// TIA Portal V18 export
FUNCTION_BLOCK "Scen2_Diag"   // FB2, FBD
TITLE = demonstrates on one variable how to generate an Alarm for HMI
   VAR_INPUT
      ID : DInt;
      Port : Int;
      EV_ID : C_Alarm_s;
   END_VAR
   VAR_OUTPUT
      Error : Bool;
      Status : Word;
      DiagDeviceFB : "LIOLink_typeDiagnostics";
   END_VAR
   VAR
      Ret : Int;
      timestamp : Date_And_Time;
      data { S7_SetPoint := 'True'} : "LIOLink_3RB24_typeAll";
      IO_LINK_3RB24_300_400_Instance { S7_SetPoint := 'True'} : "LIOLink_3RB24";
      REQ : Bool;
      Done : Bool;
      busy : Bool;
      M3 : Bool;
      M2 : Bool;
      M1 : Bool;
      error_1 : Bool;
      IEC_Timer_0_Instance { S7_SetPoint := 'True'} : TP;
   END_VAR
   VAR_TEMP
      Error_temp_1 : Bool;
      Error_temp_2 : Bool;
      status_1 : DWord;
      status_2 : DWord;
   END_VAR
   VAR_TEMP   // added for the SCL form of the ladder/FBD networks
      _w1 : Bool;
   END_VAR
BEGIN

REGION Network 1
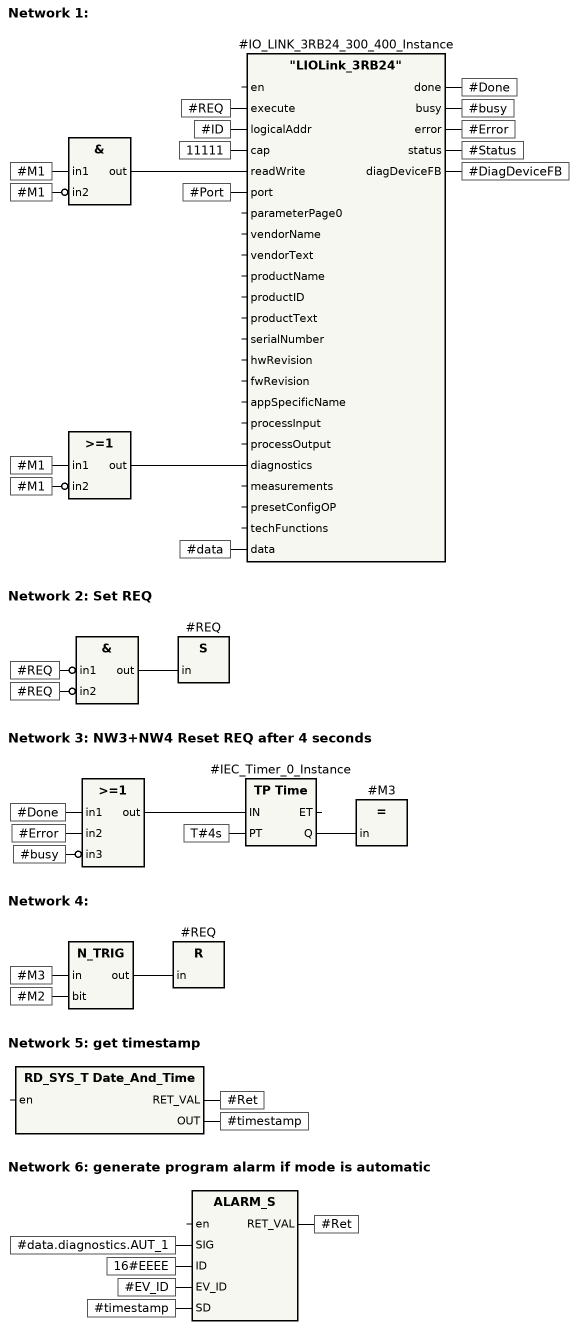
   #IO_LINK_3RB24_300_400_Instance(execute := #REQ,   // "LIOLink_3RB24"
                           logicalAddr := #ID,
                           cap := 11111,
                           readWrite := #M1 AND NOT #M1,
                           port := #Port,
                           diagnostics := #M1 OR NOT #M1,
                           data := #data,
                           done => #Done,
                           busy => #busy,
                           error => #Error,
                           status => #Status,
                           diagDeviceFB => #DiagDeviceFB);
END_REGION

REGION Network 2: Set REQ
   IF NOT #REQ AND NOT #REQ THEN #REQ := TRUE; END_IF;
END_REGION

REGION Network 3: NW3+NW4 Reset REQ after 4 seconds
   #IEC_Timer_0_Instance.TP(IN := #Done OR #Error OR NOT #busy, PT := T#4s);
   #M3 := #IEC_Timer_0_Instance.Q;
END_REGION

REGION Network 4
   #_w1 := NOT #M3 AND #M2;   // falling edge
   #M2 := #M3;
   IF #_w1 THEN #REQ := FALSE; END_IF;
END_REGION

REGION Network 5: get timestamp
   #Ret := RD_SYS_T(OUT => #timestamp);
END_REGION

REGION Network 6: generate program alarm if mode is automatic
   #Ret := ALARM_S(SIG := #data.diagnostics.AUT_1, ID := 16#EEEE, EV_ID := #EV_ID, SD := #timestamp);
END_REGION
END_FUNCTION_BLOCK
